// TwinCAT 3 PLC project PLC1
// ProgramVersion: 3.1.4020.4
// libraries:
//   Tc2_MC2, * (Beckhoff Automation GmbH)
//   Tc2_Standard, * (Beckhoff Automation GmbH)
//   Tc2_System, * (Beckhoff Automation GmbH)
//   Tc3_Module, * (Beckhoff Automation GmbH)
// project tree:
//   GVLs/ myGVL.TcGVL
//   / PlcTask.TcTTO (not stored)
//   POUs/ MAIN.TcPOU
// real-time tasks:
//   TASK PlcTask: cycle T#10ms, priority 20, ADS port 350
// motion (NC):
//   TASK NC-Task 1 SAF: cycle T#2ms, priority 4, ADS port 501
//   TASK NC-Task 1 SVB: cycle T#10ms, priority 8, ADS port 511
//   AXIS Axis 1 (id 1)
//     Dynamic: AccelerationMaximum=20000, DecelerationMaximum=20000, Acceleration=10000, Deceleration=10000, Jerk=219069
//     Velo: Maximum=1000
//     OtherSettings: AllowMotionCmdToSlave=true
//     encoder EncType=19
//       EncPara: ScaleFactorNumerator=90, ScaleFactorDenominator=65536, MaxCount=#xffffffff
//         SoftEndMinControl: Enable=true, Range=100
//         SoftEndMaxControl: Enable=true, Range=900
//         Inc: RefSearchInverse=true, RefMode=5
//     drive DrvType=16
//       DrvPara: MaxCount=#xffffffff, DriveControlDWord=#x00000100
//         Analog: VeloReferenz=1100
//         TimeComp: TaskDelayCycles=1
//     controller CtrType=1
//       CtrPara: PriorControlFactor=1
//         Observer: BandWidth=20
//   AXIS Axis 2 (id 2)
//     Dynamic: AccelerationMaximum=20000, DecelerationMaximum=20000, Acceleration=10000, Deceleration=10000, Jerk=219069
//     Velo: Maximum=1000
//     OtherSettings: AllowMotionCmdToSlave=true
//     encoder EncType=19
//       EncPara: ScaleFactorNumerator=90, ScaleFactorDenominator=65536, MaxCount=#xffffffff
//         SoftEndMinControl: Enable=true, Range=100
//         SoftEndMaxControl: Enable=true, Range=900
//         Inc: RefSearchInverse=true, RefMode=5
//     drive DrvType=16
//       DrvPara: MaxCount=#xffffffff, DriveControlDWord=#x00000100
//         Analog: VeloReferenz=1100
//         TimeComp: TaskDelayCycles=1
//     controller CtrType=1
//       CtrPara: PriorControlFactor=1
//         Observer: BandWidth=20
// I/O:
//   DEVICE NIC, AmsNetId 192.168.2.43.2.1
//     Ctr1 [CMMP-AS V4p0 CiA402]
//     Ctr2 [CMMP-AS V4p0 CiA402]
// variable links:
//   NC-Task 1 SAF/Axes/Axis 1 <-> NIC/Ctr1
//     Drive/Inputs/In/nDataIn1 <-> Inputs_1/Following_Error_Actual_Value
//     Drive/Inputs/In/nDcOutputTime <-> InfoData/DcOutputShift
//     Drive/Inputs/In/nState1 <-> Inputs/Statusword
//     Drive/Inputs/In/nState2 <-> Inputs/Statusword @bit 8
//     Drive/Inputs/In/nState4 @bit 1 <-> WcState/InputToggle
//     Drive/Inputs/In/nState4 <-> WcState/WcState
//     Drive/Outputs/Out/nCtrl1 <-> Outputs/Controlword
//     Drive/Outputs/Out/nCtrl2 <-> Outputs/Controlword @bit 8
//     Drive/Outputs/Out/nDataOut1 <-> Outputs/IP_Data_Record
//     Enc/Inputs/In/nDataIn1 <-> Inputs/Position_Actual_Value
//     Enc/Inputs/In/nDcInputTime <-> InfoData/DcInputShift
//     Enc/Inputs/In/nState4 @bit 1 <-> WcState/InputToggle
//     Enc/Inputs/In/nState4 <-> WcState/WcState
//   NC-Task 1 SAF/Axes/Axis 2 <-> NIC/Ctr2
//     Drive/Inputs/In/nDataIn1 <-> Inputs_1/Following_Error_Actual_Value
//     Drive/Inputs/In/nDcOutputTime <-> InfoData/DcOutputShift
//     Drive/Inputs/In/nState1 <-> Inputs/Statusword
//     Drive/Inputs/In/nState2 <-> Inputs/Statusword @bit 8
//     Drive/Inputs/In/nState4 @bit 1 <-> WcState/InputToggle
//     Drive/Inputs/In/nState4 <-> WcState/WcState
//     Drive/Outputs/Out/nCtrl1 <-> Outputs/Controlword
//     Drive/Outputs/Out/nCtrl2 <-> Outputs/Controlword @bit 8
//     Drive/Outputs/Out/nDataOut1 <-> Outputs/IP_Data_Record
//     Enc/Inputs/In/nDataIn1 <-> Inputs/Position_Actual_Value
//     Enc/Inputs/In/nDcInputTime <-> InfoData/DcInputShift
//     Enc/Inputs/In/nState4 @bit 1 <-> WcState/InputToggle
//     Enc/Inputs/In/nState4 <-> WcState/WcState
//   PLC1/PLC1 Instance <-> NC-Task 1 SAF/Axes/Axis 1
//     PlcTask Inputs/myGVL.Axis1.NcToPlc <-> Outputs/ToPlc
//     PlcTask Outputs/myGVL.Axis1.PlcToNc <-> Inputs/FromPlc
//   PLC1/PLC1 Instance <-> NC-Task 1 SAF/Axes/Axis 2
//     PlcTask Inputs/myGVL.Axis2.NcToPlc <-> Outputs/ToPlc
//     PlcTask Outputs/myGVL.Axis2.PlcToNc <-> Inputs/FromPlc

// ---- GVLs/myGVL.TcGVL
{attribute 'qualified_only'}
VAR_GLOBAL
	Axis1 : AXIS_REF;
	Axis2 : AXIS_REF;
END_VAR

// ---- POUs/MAIN.TcPOU
PROGRAM MAIN
VAR
	fbPower: MC_Power;
	EnableAxis1 : BOOL;
	AxisEnabled : BOOL;
	Error : BOOL;
	ErrorID: UDINT;
	
	fbJog: MC_Jog;	
	JogForwardPB : BOOL;
	JogBackwardPB : BOOL;
	

	fbHome: MC_Home;
	HomePB: BOOL;
	
	
	fbReadStatus: MC_ReadStatus;
	AxisStatus: ST_AxisStatus;
	
	JogError: BOOL;
	JogErrorID: UDINT;
	
	
	fbMoveAbsolute: MC_MoveAbsolute;
	MoveExecute: BOOL;
	MovePosition: LREAL;
END_VAR

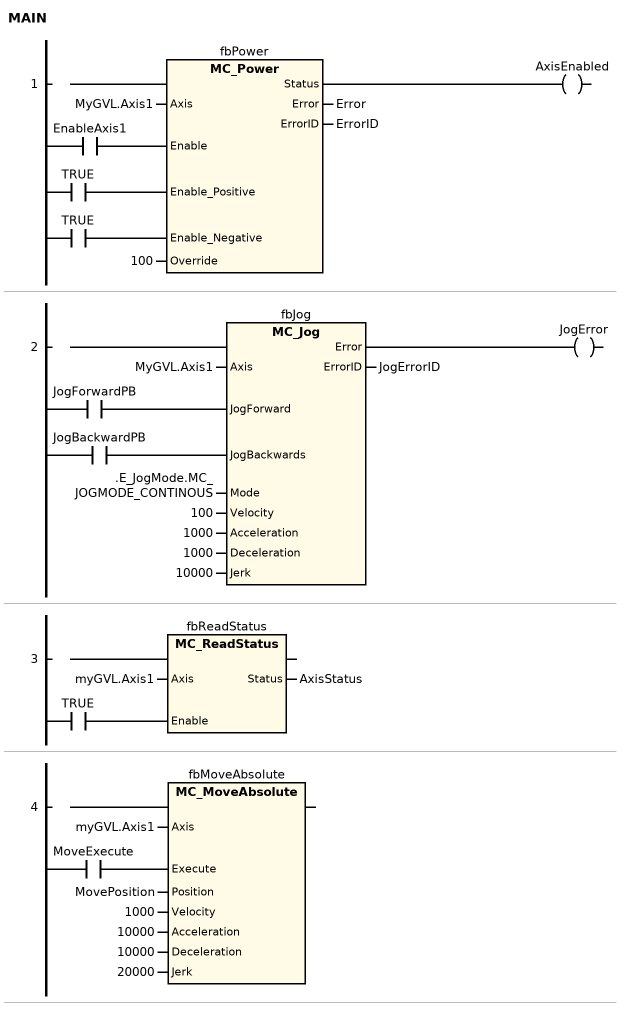
// NETWORK 1
fbPower(
    Axis := MyGVL.Axis1,
    Enable := EnableAxis1,
    Enable_Positive := TRUE,
    Enable_Negative := TRUE,
    Override := 100,
    Error => Error,
    ErrorID => ErrorID); // MC_Power
AxisEnabled := fbPower.Status;

// NETWORK 2
fbJog(
    Axis := MyGVL.Axis1,
    JogForward := JogForwardPB,
    JogBackwards := JogBackwardPB,
    Mode := .E_JogMode.MC_JOGMODE_CONTINOUS,
    Velocity := 100,
    Acceleration := 1000,
    Deceleration := 1000,
    Jerk := 10000,
    Error => JogError,
    ErrorID => JogErrorID); // MC_Jog

// NETWORK 3
fbReadStatus(Axis := myGVL.Axis1, Enable := TRUE, Status => AxisStatus); // MC_ReadStatus

// NETWORK 4
fbMoveAbsolute(
    Axis := myGVL.Axis1,
    Execute := MoveExecute,
    Position := MovePosition,
    Velocity := 1000,
    Acceleration := 10000,
    Deceleration := 10000,
    Jerk := 20000); // MC_MoveAbsolute

END_PROGRAM
